KUKA KRL program: RoofInterrupt.src

&ACCESS RV1
&REL 6
&PARAM EDITMASK = *
&PARAM TEMPLATE = C:\KRC\Roboter\Template\vorgabe
DEF RoofInterrupt( )
;************************************************
;              CNC Robotics Ltd
;              www.cncrobotics.co.uk
;************************************************
;     Contact: helpdesk@cncrobotics.co.uk
;     Date: 25/09/23
;     Version: 0.13.38
;************************************************
; Description: Interrup to control what happens in
; the event of a fault.
;************************************************

BRAKE

bRoofInterrupt = FALSE

END
